FUNCTION_BLOCK StateAborted EXTENDS _AbstractState
VAR
	_bInternalLock: BOOL;
END_VAR

(*
Executed when the state is entered.  
Provides a hook for defining state-specific behavior to be performed during the transition into this state.
*)
METHOD PROTECTED OnEntry
_ctx.sHmiStatusText := 'Aborted: Something bad happened!';
END_METHOD

END_FUNCTION_BLOCK

(* stored: Version 1.1.0.1
   POU StateAborted: Id {746106d1-75ed-4c27-8afa-f94a3812261d}, SpecialFunc None
   Method OnEntry: Id {57cd4973-d9f8-4598-9f13-9b3abdf2da09} *)
